{attribute addProperty BoxType "EL5101-0000-0001"}
{attribute addProperty Id "InputsAT %I*Inputs_6F37F4E44050OutputsAT %Q*Outputs_4D4E89362430WcStateAT %I*WcState_98A4DF7520.250InfoDataAT %I*InfoData_BC63D37F80100"}
{attribute addProperty CRC "1890814869"}
{attribute addProperty SizeInBites "146"}
{attribute addProperty SizeInBytes "18.25"}
TYPE EL5101_38C6EF5E :
STRUCT
	{attribute addProperty Name "Inputs"}
	Inputs : Inputs_6F37F4E4;
	{attribute addProperty Name "Outputs"}
	Outputs : Outputs_4D4E8936;
	{attribute addProperty Name "WcState"}
	WcState : WcState_98A4DF75;
	{attribute addProperty Name "InfoData"}
	InfoData : InfoData_BC63D37F;
END_STRUCT
END_TYPE

(* stored: Version 1.2.0.0, ProductVersion 3.1.4024.9
   DUT EL5101_38C6EF5E: Id {b4e18192-0571-4498-8f09-ce2e348955ad} *)
